% RSLogix 500 project 3 CHEMICAL TANK MIXING CONTROL.RSS, saved by version 8.30.00.16 %
PROJECT "UNTITLED"    % processor: Bul.1763 MicroLogix 1100 Series B %

PROGRAM FILES
  LAD 2   4 rungs

DATA FILES
  O0 OUTPUT  4 elements
  I1 INPUT  6 elements
  S2 STATUS  66 elements
  B3 BINARY  1 elements
  T4 TIMER  1 elements
  C5 COUNTER  1 elements
  R6 CONTROL  1 elements
  N7 INTEGER  1 elements
  F8 FLOAT  1 elements

LADDER 2
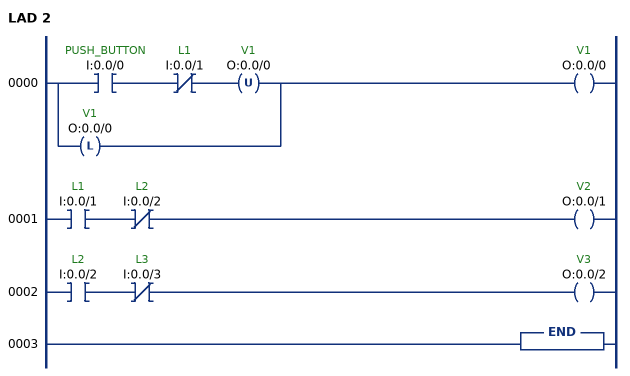
% Rung: 0 %  % edit flag set %
SOR BST XIC I:0.0/0 XIO I:0.0/1 OTU O:0.0/0 NXB OTL O:0.0/0 BND OTE O:0.0/0 EOR
%   I:0.0/0  PUSH_BUTTON %
%   I:0.0/1  L1 %
%   O:0.0/0  V1 %
% Rung: 1 %
SOR XIC I:0.0/1 XIO I:0.0/2 OTE O:0.0/1 EOR
%   I:0.0/1  L1 %
%   I:0.0/2  L2 %
%   O:0.0/1  V2 %
% Rung: 2 %
SOR XIC I:0.0/2 XIO I:0.0/3 OTE O:0.0/2 EOR
%   I:0.0/2  L2 %
%   I:0.0/3  L3 %
%   O:0.0/2  V3 %
% Rung: 3 %
SOR END EOR
